% RSLogix 500 project Water Tank.RSS, saved by version 8.30.00.16 %
PROJECT "UNTITLED"    % processor: Bul.1763 MicroLogix 1100 Series B %

PROGRAM FILES
  LAD 2 "MAIN"  4 rungs
  LAD 3 "DIGITAL IO"  7 rungs
  LAD 4 "CONTROLS"  10 rungs
  LAD 5 "ALARMS"  7 rungs

DATA FILES
  O0 OUTPUT  5 elements
  I1 INPUT  7 elements
  S2 STATUS  66 elements
  B3 BINARY  2 elements
  T4 TIMER  4 elements
  C5 COUNTER  1 elements
  R6 CONTROL  1 elements
  N7 INTEGER  1 elements
  F8 FLOAT  1 elements

LADDER 2 "MAIN"
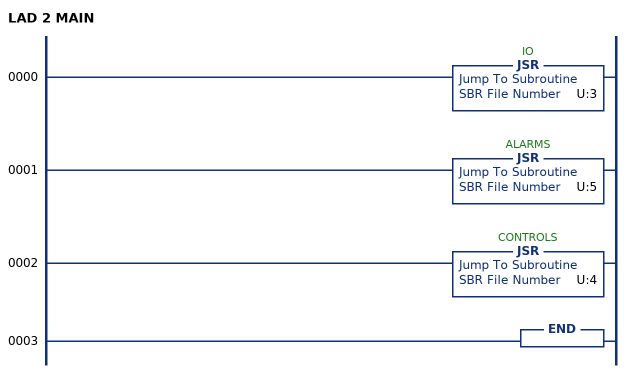
% Rung: 0 %
SOR JSR U:3 EOR
%   U:3  "IO" %
% Rung: 1 %
SOR JSR U:5 EOR
%   U:5  "ALARMS" %
% Rung: 2 %
SOR JSR U:4 EOR
%   U:4  "CONTROLS" %
% Rung: 3 %
SOR END EOR

LADDER 3 "DIGITAL IO"
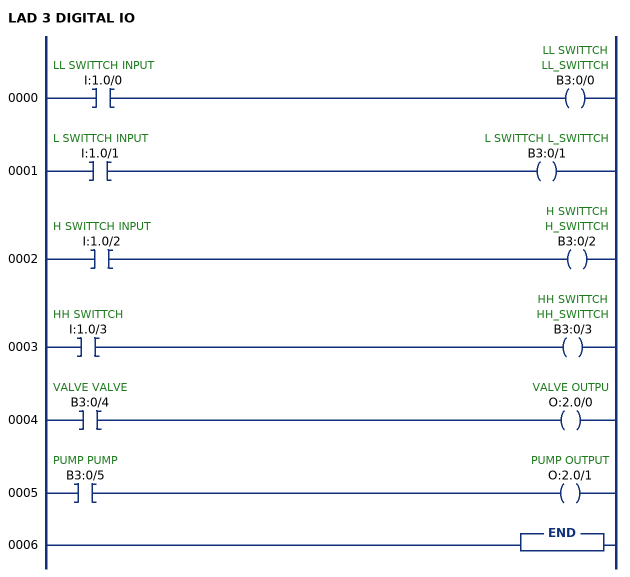
% Rung: 0 %
SOR XIC I:1.0/0 OTE B3:0/0 EOR
%   I:1.0/0  "LL SWITTCH INPUT" %
%   B3:0/0  LL_SWITTCH  "LL SWITTCH" %
% Rung: 1 %
SOR XIC I:1.0/1 OTE B3:0/1 EOR
%   I:1.0/1  "L SWITTCH INPUT" %
%   B3:0/1  L_SWITTCH  "L SWITTCH" %
% Rung: 2 %
SOR XIC I:1.0/2 OTE B3:0/2 EOR
%   I:1.0/2  "H SWITTCH INPUT" %
%   B3:0/2  H_SWITTCH  "H SWITTCH" %
% Rung: 3 %
SOR XIC I:1.0/3 OTE B3:0/3 EOR
%   I:1.0/3  "HH SWITTCH" %
%   B3:0/3  HH_SWITTCH  "HH SWITTCH" %
% Rung: 4 %
SOR XIC B3:0/4 OTE O:2.0/0 EOR
%   B3:0/4  VALVE  "VALVE" %
%   O:2.0/0  "VALVE OUTPU" %
% Rung: 5 %
SOR XIC B3:0/5 OTE O:2.0/1 EOR
%   B3:0/5  PUMP  "PUMP" %
%   O:2.0/1  "PUMP OUTPUT" %
% Rung: 6 %
SOR END EOR

LADDER 4 "CONTROLS"
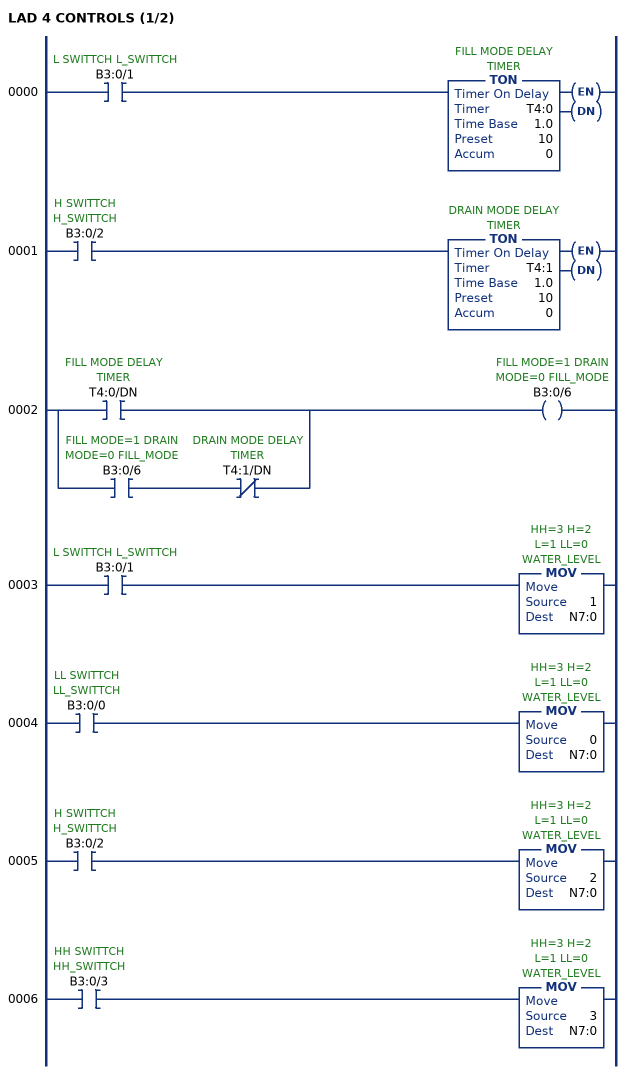
% Rung: 0 %
SOR XIC B3:0/1 TON T4:0 1.0 10 0 EOR
%   B3:0/1  L_SWITTCH  "L SWITTCH" %
%   T4:0  "FILL MODE DELAY TIMER" %
% Rung: 1 %
SOR XIC B3:0/2 TON T4:1 1.0 10 0 EOR
%   B3:0/2  H_SWITTCH  "H SWITTCH" %
%   T4:1  "DRAIN MODE DELAY TIMER" %
% Rung: 2 %
SOR BST XIC T4:0/DN NXB XIC B3:0/6 XIO T4:1/DN BND OTE B3:0/6 EOR
%   T4:0  "FILL MODE DELAY TIMER" %
%   B3:0/6  FILL_MODE  "FILL MODE=1 DRAIN MODE=0" %
%   T4:1  "DRAIN MODE DELAY TIMER" %
% Rung: 3 %
SOR XIC B3:0/1 MOV 1 N7:0 EOR
%   B3:0/1  L_SWITTCH  "L SWITTCH" %
%   N7:0  WATER_LEVEL  "HH=3 H=2 L=1 LL=0" %
% Rung: 4 %
SOR XIC B3:0/0 MOV 0 N7:0 EOR
%   B3:0/0  LL_SWITTCH  "LL SWITTCH" %
%   N7:0  WATER_LEVEL  "HH=3 H=2 L=1 LL=0" %
% Rung: 5 %
SOR XIC B3:0/2 MOV 2 N7:0 EOR
%   B3:0/2  H_SWITTCH  "H SWITTCH" %
%   N7:0  WATER_LEVEL  "HH=3 H=2 L=1 LL=0" %
% Rung: 6 %
SOR XIC B3:0/3 MOV 3 N7:0 EOR
%   B3:0/3  HH_SWITTCH  "HH SWITTCH" %
%   N7:0  WATER_LEVEL  "HH=3 H=2 L=1 LL=0" %

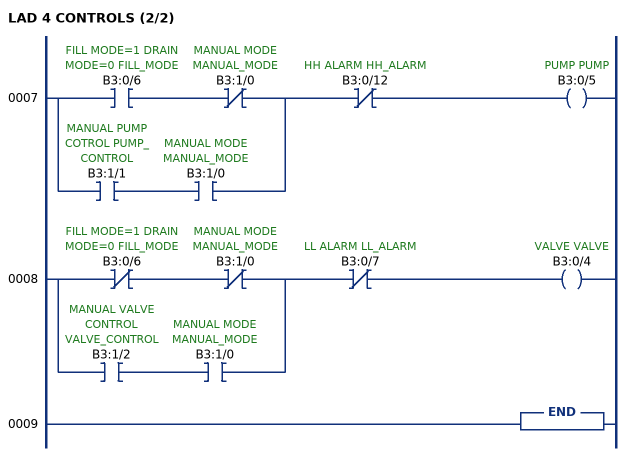
% Rung: 7 %
SOR BST XIC B3:0/6 XIO B3:1/0 NXB XIC B3:1/1 XIC B3:1/0 BND XIO B3:0/12 OTE B3:0/5 EOR
%   B3:0/6  FILL_MODE  "FILL MODE=1 DRAIN MODE=0" %
%   B3:1/0  MANUAL_MODE  "MANUAL MODE" %
%   B3:1/1  PUMP_CONTROL  "MANUAL PUMP COTROL" %
%   B3:0/12  HH_ALARM  "HH ALARM" %
%   B3:0/5  PUMP  "PUMP" %
% Rung: 8 %
SOR BST XIO B3:0/6 XIO B3:1/0 NXB XIC B3:1/2 XIC B3:1/0 BND XIO B3:0/7 OTE B3:0/4 EOR
%   B3:0/6  FILL_MODE  "FILL MODE=1 DRAIN MODE=0" %
%   B3:1/0  MANUAL_MODE  "MANUAL MODE" %
%   B3:1/2  VALVE_CONTROL  "MANUAL VALVE CONTROL" %
%   B3:0/7  LL_ALARM  "LL ALARM" %
%   B3:0/4  VALVE  "VALVE" %
% Rung: 9 %
SOR END EOR

LADDER 5 "ALARMS"
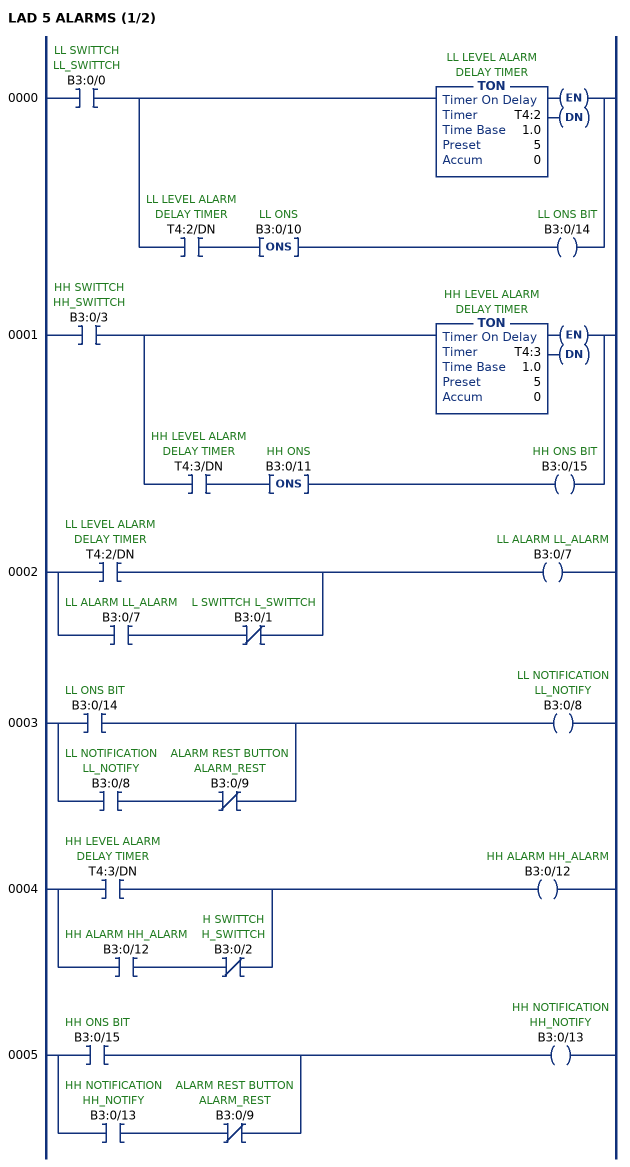
% Rung: 0 %
SOR XIC B3:0/0 BST TON T4:2 1.0 5 0 NXB XIC T4:2/DN ONS B3:0/10 OTE B3:0/14 BND EOR
%   B3:0/0  LL_SWITTCH  "LL SWITTCH" %
%   T4:2  "LL LEVEL ALARM DELAY TIMER" %
%   B3:0/10  "LL ONS" %
%   B3:0/14  "LL ONS BIT" %
% Rung: 1 %
SOR XIC B3:0/3 BST TON T4:3 1.0 5 0 NXB XIC T4:3/DN ONS B3:0/11 OTE B3:0/15 BND EOR
%   B3:0/3  HH_SWITTCH  "HH SWITTCH" %
%   T4:3  "HH LEVEL ALARM DELAY TIMER" %
%   B3:0/11  "HH ONS" %
%   B3:0/15  "HH ONS BIT" %
% Rung: 2 %
SOR BST XIC T4:2/DN NXB XIC B3:0/7 XIO B3:0/1 BND OTE B3:0/7 EOR
%   T4:2  "LL LEVEL ALARM DELAY TIMER" %
%   B3:0/7  LL_ALARM  "LL ALARM" %
%   B3:0/1  L_SWITTCH  "L SWITTCH" %
% Rung: 3 %
SOR BST XIC B3:0/14 NXB XIC B3:0/8 XIO B3:0/9 BND OTE B3:0/8 EOR
%   B3:0/14  "LL ONS BIT" %
%   B3:0/8  LL_NOTIFY  "LL NOTIFICATION" %
%   B3:0/9  ALARM_REST  "ALARM REST BUTTON" %
% Rung: 4 %
SOR BST XIC T4:3/DN NXB XIC B3:0/12 XIO B3:0/2 BND OTE B3:0/12 EOR
%   T4:3  "HH LEVEL ALARM DELAY TIMER" %
%   B3:0/12  HH_ALARM  "HH ALARM" %
%   B3:0/2  H_SWITTCH  "H SWITTCH" %
% Rung: 5 %
SOR BST XIC B3:0/15 NXB XIC B3:0/13 XIO B3:0/9 BND OTE B3:0/13 EOR
%   B3:0/15  "HH ONS BIT" %
%   B3:0/13  HH_NOTIFY  "HH NOTIFICATION" %
%   B3:0/9  ALARM_REST  "ALARM REST BUTTON" %

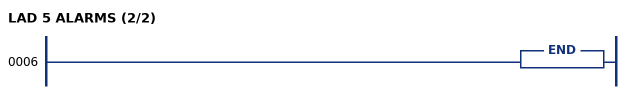
% Rung: 6 %
SOR END EOR

DATA TABLE (non-zero values as saved)
DATA T4
% .PRE .ACC %
% T4:0 % 10 0
% T4:1 % 10 0
% T4:2 % 5 0
% T4:3 % 5 0
